FUNCTION_BLOCK FB_RiseEdgeCheck
VAR
	// last value
	m_lastValue :BOOL:=false;
END_VAR

METHOD check : BOOL
VAR_INPUT
	input :BOOL;
END_VAR
IF NOT(m_lastValue) AND input THEN
	check := TRUE;
ELSE
	check :=FALSE;
END_IF

m_lastValue := input;
END_METHOD

METHOD reset : BOOL
m_lastValue := false;
END_METHOD

END_FUNCTION_BLOCK

(* stored: Version 1.1.0.1, ProductVersion 3.1.4024.12
   POU FB_RiseEdgeCheck: Id {54f969e7-bfb8-4c92-8c48-75d0e1f9ed72}, SpecialFunc None
   Method check: Id {980b320f-3ebe-4bf1-98f5-ddf6a02c6d3f}
   Method reset: Id {d17487e9-29ea-4ea4-bd4c-f5339a37b6fc} *)
